Fanuc KAREL source: kt00513.KL

PROGRAM KT00513
%STACKSIZE=65535
%PRIORITY=65535
%NOLOCKGROUP
VAR
P1 : XYZWPREXT
P2 : POSITION
OUT : BOOLEAN
BEGIN
P1.X=1.0
-- UNRESOLVED_PC line 9 opcodes [49 7E 49 AC 23] marker_code=20
END KT00513
